# EPICS substitutions: motorSim/motorSimApp/Db/motorSim.substitutions
file "db/motorAsyn.db"
{
pattern
{P,            N,  M,           DTYP,        PORT,       ADDR,  DESC,          EGU,      DIR,  VELO,  VBAS,  ACCL,  BDST,  BVEL,  BACC,  MRES,  PREC,  DHLM,  DLLM,  INIT}
{"$(PREFIX)",  1,  "Mtr$(N)",  "asynMotor",  "$(MPORT)",  0,     "motor $(N)",  degrees,  Pos,  1,     .1,    .2,    0,     1,     .2,    0.01,  5,     100,   -100,  ""}
{"$(PREFIX)",  2,  "Mtr$(N)",  "asynMotor",  "$(MPORT)",  1,     "motor $(N)",  degrees,  Pos,  1,     .1,    .2,    0,     1,     .2,    0.01,  5,     100,   -100,  ""}
{"$(PREFIX)",  3,  "Mtr$(N)",  "asynMotor",  "$(MPORT)",  2,     "motor $(N)",  degrees,  Pos,  1,     .1,    .2,    0,     1,     .2,    0.01,  5,     100,   -100,  ""}
{"$(PREFIX)",  4,  "Mtr$(N)",  "asynMotor",  "$(MPORT)",  3,     "motor $(N)",  degrees,  Pos,  1,     .1,    .2,    0,     1,     .2,    0.01,  5,     100,   -100,  ""}
{"$(PREFIX)",  5,  "Mtr$(N)",  "asynMotor",  "$(MPORT)",  4,     "motor $(N)",  degrees,  Pos,  1,     .1,    .2,    0,     1,     .2,    0.01,  5,     100,   -100,  ""}
{"$(PREFIX)",  6,  "Mtr$(N)",  "asynMotor",  "$(MPORT)",  5,     "motor $(N)",  degrees,  Pos,  1,     .1,    .2,    0,     1,     .2,    0.01,  5,     100,   -100,  ""}
{"$(PREFIX)",  7,  "Mtr$(N)",  "asynMotor",  "$(MPORT)",  6,     "motor $(N)",  degrees,  Pos,  1,     .1,    .2,    0,     1,     .2,    0.01,  5,     100,   -100,  ""}
{"$(PREFIX)",  8,  "Mtr$(N)",  "asynMotor",  "$(MPORT)",  7,     "motor $(N)",  degrees,  Pos,  1,     .1,    .2,    0,     1,     .2,    0.01,  5,     100,   -100,  ""}
}
